KUKA KRL program: Screwing_Demo.src, Screwing_Demo.dat

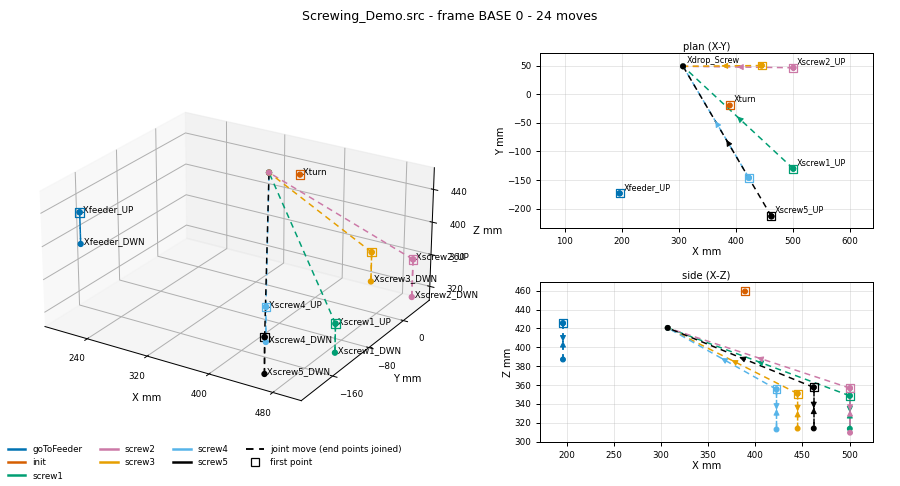
[picture p0: tool path of Screwing_Demo.src in frame BASE 0, 24 of 28 moves have a stored position in this frame; points joined in program order, loops and branches not executed]
--- Screwing_Demo.src ---
&ACCESS RVP
&REL 1
&PARAM DISKPATH = KRC:\R1\Program
DEF Screwing_Demo( )
INTERRUPT DECL 3 WHEN aiVacuumInput < 0.230 DO screwDropInterrupt()
;FOLD INI;%{PE}
  ;FOLD BASISTECH INI
    GLOBAL INTERRUPT DECL 3 WHEN $STOPMESS==TRUE DO IR_STOPM ( )
    INTERRUPT ON 3
    BAS (#INITMOV,0 )
  ;ENDFOLD (BASISTECH INI)
;FOLD SPOTTECH INI
USERSPOT(#INIT)
;ENDFOLD (SPOTTECH INI)
;FOLD GRIPPERTECH INI
USER_GRP(0,DUMMY,DUMMY,GDEFAULT)
;ENDFOLD (GRIPPERTECH INI)
  ;FOLD USER INI
    ;Make your modifications here

  ;ENDFOLD (USER INI)
;ENDFOLD (INI)
;FOLD PTP HOME  Vel= 100 % DEFAULT;%{PE}%MKUKATPBASIS,%CMOVE,%VPTP,%P 1:PTP, 2:HOME, 3:, 5:100, 7:DEFAULT
$BWDSTART = FALSE
PDAT_ACT=PDEFAULT
FDAT_ACT=FHOME
BAS (#PTP_PARAMS,100 )
$H_POS=XHOME
PTP  XHOME
;ENDFOLD
num_state_machine = 1
LOOP
 SWITCH num_state_machine
  CASE init_state
    init()
  CASE screw1_state
   resetOutputs()
   goToFeeder()
   screw1()
  CASE screw2_state
   resetOutputs()
   goToFeeder()
   screw2()
  CASE screw3_state
   resetOutputs()
   goToFeeder()
   screw3()
  CASE screw4_state
   resetOutputs()
   goToFeeder()
   screw4()
  CASE screw5_state
   resetOutputs()
   goToFeeder()
   screw5()
  CASE error_state
   EXIT
 ENDSWITCH
ENDLOOP
END
DEF screwingProcess()
 $ACC.CP = 1
 $VEL.CP = 1
 INTERRUPT ON
 LIN_REL { Z - 15}
 WAIT FOR TRUE
END
DEF goToFeeder()
;FOLD PTP feeder_UP Vel=100 % PDAT2 Tool[1] Base[0];%{PE}%R 8.3.40,%MKUKATPBASIS,%CMOVE,%VPTP,%P 1:PTP, 2:feeder_UP, 3:, 5:100, 7:PDAT2
$BWDSTART=FALSE
PDAT_ACT=PPDAT2
FDAT_ACT=Ffeeder_UP
BAS(#PTP_PARAMS,100)
PTP Xfeeder_UP
;ENDFOLD
 setVel()
;FOLD PTP feeder_DWN Vel=100 % PDAT3 Tool[1] Base[0];%{PE}%R 8.3.40,%MKUKATPBASIS,%CMOVE,%VPTP,%P 1:PTP, 2:feeder_DWN, 3:, 5:100, 7:PDAT3
$BWDSTART=FALSE
PDAT_ACT=PPDAT3
FDAT_ACT=Ffeeder_DWN
BAS(#PTP_PARAMS,100)
PTP Xfeeder_DWN
;ENDFOLD
 Vacuum_ON = TRUE
 ANIN ON vacuumValue = 1.0 * aiVacuumInput
 WAIT FOR vacuumValue >= 0.23
 ANIN OFF aiVacuumInput
;FOLD PTP feeder_UP Vel=100 % PDAT4 Tool[1] Base[0];%{PE}%R 8.3.40,%MKUKATPBASIS,%CMOVE,%VPTP,%P 1:PTP, 2:feeder_UP, 3:, 5:100, 7:PDAT4
$BWDSTART=FALSE
PDAT_ACT=PPDAT4
FDAT_ACT=Ffeeder_UP
BAS(#PTP_PARAMS,100)
PTP Xfeeder_UP
;ENDFOLD
END
DEF screwInterruptOK()
 INTERRUPT OFF
 BRAKE
 LIN $POS_INT
 RESUME
END
DEF screwInterruptNOK()
 INTERRUPT OFF
 BRAKE
 LIN $POS_INT
 RESUME
END
DEF setVel()
 $OV_PRO = 10
 $ACC.CP = 2
 $VEL.CP = 2
END
DEF setPathVel()
 $OV_PRO = 60
END
DEF init()
 setPathVel()
;FOLD PTP turn Vel=100 % PDAT1 Tool[1] Base[0];%{PE}%R 8.3.40,%MKUKATPBASIS,%CMOVE,%VPTP,%P 1:PTP, 2:turn, 3:, 5:100, 7:PDAT1
$BWDSTART=FALSE
PDAT_ACT=PPDAT1
FDAT_ACT=Fturn
BAS(#PTP_PARAMS,100)
PTP Xturn
;ENDFOLD
 num_state_machine = screw1_state
END
DEF resetOutputs()
 doResetProg = TRUE
 WAIT SEC 0.024
 doStartScrewing = FALSE
 doResetProg = FALSE
END
DEF screw1()
INTERRUPT DECL 1 WHEN diScrewOK DO screwInterruptOK()
INTERRUPT DECL 2 WHEN diScrewNOK DO screwInterruptNOK()
setPathVel()
;FOLD PTP screw1_UP Vel=100 % PDAT7 Tool[1] Base[0];%{PE}%R 8.3.40,%MKUKATPBASIS,%CMOVE,%VPTP,%P 1:PTP, 2:screw1_UP, 3:, 5:100, 7:PDAT7
$BWDSTART=FALSE
PDAT_ACT=PPDAT7
FDAT_ACT=Fscrew1_UP
BAS(#PTP_PARAMS,100)
PTP Xscrew1_UP
;ENDFOLD
setVel()
;FOLD PTP screw1_DWN Vel=100 % PDAT6 Tool[1] Base[0];%{PE}%R 8.3.40,%MKUKATPBASIS,%CMOVE,%VPTP,%P 1:PTP, 2:screw1_DWN, 3:, 5:100, 7:PDAT6
$BWDSTART=FALSE
PDAT_ACT=PPDAT6
FDAT_ACT=Fscrew1_DWN
BAS(#PTP_PARAMS,100)
PTP Xscrew1_DWN
;ENDFOLD
 doStartScrewing = TRUE
 screwingProcess()
 Vacuum_ON = FALSE
setPathVel()
;FOLD PTP screw1_UP Vel=100 % PDAT8 Tool[1] Base[0];%{PE}%R 8.3.40,%MKUKATPBASIS,%CMOVE,%VPTP,%P 1:PTP, 2:screw1_UP, 3:, 5:100, 7:PDAT8
$BWDSTART=FALSE
PDAT_ACT=PPDAT8
FDAT_ACT=Fscrew1_UP
BAS(#PTP_PARAMS,100)
PTP Xscrew1_UP
;ENDFOLD
;FOLD PTP drop_Screw Vel=100 % PDAT5 Tool[1] Base[0];%{PE}%R 8.3.40,%MKUKATPBASIS,%CMOVE,%VPTP,%P 1:PTP, 2:drop_Screw, 3:, 5:100, 7:PDAT5
$BWDSTART=FALSE
PDAT_ACT=PPDAT5
FDAT_ACT=Fdrop_Screw
BAS(#PTP_PARAMS,100)
PTP Xdrop_Screw
;ENDFOLD
 num_state_machine = screw2_state
END
DEF screw2()
setPathVel()
;FOLD PTP screw2_UP Vel=100 % PDAT10 Tool[1] Base[0];%{PE}%R 8.3.40,%MKUKATPBASIS,%CMOVE,%VPTP,%P 1:PTP, 2:screw2_UP, 3:, 5:100, 7:PDAT10
$BWDSTART=FALSE
PDAT_ACT=PPDAT10
FDAT_ACT=Fscrew2_UP
BAS(#PTP_PARAMS,100)
PTP Xscrew2_UP
;ENDFOLD
setVel()
;FOLD PTP screw2_DWN Vel=100 % PDAT9 Tool[1] Base[0];%{PE}%R 8.3.40,%MKUKATPBASIS,%CMOVE,%VPTP,%P 1:PTP, 2:screw2_DWN, 3:, 5:100, 7:PDAT9
$BWDSTART=FALSE
PDAT_ACT=PPDAT9
FDAT_ACT=Fscrew2_DWN
BAS(#PTP_PARAMS,100)
PTP Xscrew2_DWN
;ENDFOLD
 doStartScrewing = TRUE
 screwingProcess()
 Vacuum_ON = FALSE
setPathVel()
;FOLD PTP screw2_UP Vel=100 % PDAT11 Tool[1] Base[0];%{PE}%R 8.3.40,%MKUKATPBASIS,%CMOVE,%VPTP,%P 1:PTP, 2:screw2_UP, 3:, 5:100, 7:PDAT11
$BWDSTART=FALSE
PDAT_ACT=PPDAT11
FDAT_ACT=Fscrew2_UP
BAS(#PTP_PARAMS,100)
PTP Xscrew2_UP
;ENDFOLD
;FOLD PTP drop_Screw Vel=100 % PDAT12 Tool[1] Base[0];%{PE}%R 8.3.40,%MKUKATPBASIS,%CMOVE,%VPTP,%P 1:PTP, 2:drop_Screw, 3:, 5:100, 7:PDAT12
$BWDSTART=FALSE
PDAT_ACT=PPDAT12
FDAT_ACT=Fdrop_Screw
BAS(#PTP_PARAMS,100)
PTP Xdrop_Screw
;ENDFOLD
 num_state_machine = screw3_state
END
DEF screw3()
 setPathVel()
;FOLD PTP screw3_UP Vel=100 % PDAT13 Tool[1] Base[0];%{PE}%R 8.3.40,%MKUKATPBASIS,%CMOVE,%VPTP,%P 1:PTP, 2:screw3_UP, 3:, 5:100, 7:PDAT13
$BWDSTART=FALSE
PDAT_ACT=PPDAT13
FDAT_ACT=Fscrew3_UP
BAS(#PTP_PARAMS,100)
PTP Xscrew3_UP
;ENDFOLD
 setVel()
;FOLD PTP screw3_DWN Vel=100 % PDAT14 Tool[1] Base[0];%{PE}%R 8.3.40,%MKUKATPBASIS,%CMOVE,%VPTP,%P 1:PTP, 2:screw3_DWN, 3:, 5:100, 7:PDAT14
$BWDSTART=FALSE
PDAT_ACT=PPDAT14
FDAT_ACT=Fscrew3_DWN
BAS(#PTP_PARAMS,100)
PTP Xscrew3_DWN
;ENDFOLD
 doStartScrewing = TRUE
 screwingProcess()
 Vacuum_ON = FALSE
 setPathVel()
;FOLD PTP screw3_UP Vel=100 % PDAT15 Tool[1] Base[0];%{PE}%R 8.3.40,%MKUKATPBASIS,%CMOVE,%VPTP,%P 1:PTP, 2:screw3_UP, 3:, 5:100, 7:PDAT15
$BWDSTART=FALSE
PDAT_ACT=PPDAT15
FDAT_ACT=Fscrew3_UP
BAS(#PTP_PARAMS,100)
PTP Xscrew3_UP
;ENDFOLD
;FOLD PTP drop_Screw Vel=100 % PDAT16 Tool[1] Base[0];%{PE}%R 8.3.40,%MKUKATPBASIS,%CMOVE,%VPTP,%P 1:PTP, 2:drop_Screw, 3:, 5:100, 7:PDAT16
$BWDSTART=FALSE
PDAT_ACT=PPDAT16
FDAT_ACT=Fdrop_Screw
BAS(#PTP_PARAMS,100)
PTP Xdrop_Screw
;ENDFOLD
 num_state_machine = screw4_state
END
DEF screw4()
 setPathVel()
;FOLD PTP screw4_UP Vel=100 % PDAT18 Tool[1] Base[0];%{PE}%R 8.3.40,%MKUKATPBASIS,%CMOVE,%VPTP,%P 1:PTP, 2:screw4_UP, 3:, 5:100, 7:PDAT18
$BWDSTART=FALSE
PDAT_ACT=PPDAT18
FDAT_ACT=Fscrew4_UP
BAS(#PTP_PARAMS,100)
PTP Xscrew4_UP
;ENDFOLD
 setVel()
;FOLD PTP screw4_DWN Vel=100 % PDAT17 Tool[1] Base[0];%{PE}%R 8.3.40,%MKUKATPBASIS,%CMOVE,%VPTP,%P 1:PTP, 2:screw4_DWN, 3:, 5:100, 7:PDAT17
$BWDSTART=FALSE
PDAT_ACT=PPDAT17
FDAT_ACT=Fscrew4_DWN
BAS(#PTP_PARAMS,100)
PTP Xscrew4_DWN
;ENDFOLD
 doStartScrewing = TRUE
 screwingProcess()
 Vacuum_ON = FALSE
 setPathVel()
;FOLD PTP screw4_UP Vel=100 % PDAT19 Tool[1] Base[0];%{PE}%R 8.3.40,%MKUKATPBASIS,%CMOVE,%VPTP,%P 1:PTP, 2:screw4_UP, 3:, 5:100, 7:PDAT19
$BWDSTART=FALSE
PDAT_ACT=PPDAT19
FDAT_ACT=Fscrew4_UP
BAS(#PTP_PARAMS,100)
PTP Xscrew4_UP
;ENDFOLD
;FOLD PTP drop_Screw Vel=100 % PDAT20 Tool[1] Base[0];%{PE}%R 8.3.40,%MKUKATPBASIS,%CMOVE,%VPTP,%P 1:PTP, 2:drop_Screw, 3:, 5:100, 7:PDAT20
$BWDSTART=FALSE
PDAT_ACT=PPDAT20
FDAT_ACT=Fdrop_Screw
BAS(#PTP_PARAMS,100)
PTP Xdrop_Screw
;ENDFOLD
 num_state_machine = screw5_state
END
DEF screw5()
 setPathVel()
;FOLD PTP screw5_UP Vel=100 % PDAT21 Tool[1] Base[0];%{PE}%R 8.3.40,%MKUKATPBASIS,%CMOVE,%VPTP,%P 1:PTP, 2:screw5_UP, 3:, 5:100, 7:PDAT21
$BWDSTART=FALSE
PDAT_ACT=PPDAT21
FDAT_ACT=Fscrew5_UP
BAS(#PTP_PARAMS,100)
PTP Xscrew5_UP
;ENDFOLD
 setVel()
;FOLD PTP screw5_DWN Vel=100 % PDAT22 Tool[1] Base[0];%{PE}%R 8.3.40,%MKUKATPBASIS,%CMOVE,%VPTP,%P 1:PTP, 2:screw5_DWN, 3:, 5:100, 7:PDAT22
$BWDSTART=FALSE
PDAT_ACT=PPDAT22
FDAT_ACT=Fscrew5_DWN
BAS(#PTP_PARAMS,100)
PTP Xscrew5_DWN
;ENDFOLD
 doStartScrewing = TRUE
 screwingProcess()
 Vacuum_ON = FALSE
 setPathVel()
;FOLD PTP screw5_UP Vel=100 % PDAT23 Tool[1] Base[0];%{PE}%R 8.3.40,%MKUKATPBASIS,%CMOVE,%VPTP,%P 1:PTP, 2:screw5_UP, 3:, 5:100, 7:PDAT23
$BWDSTART=FALSE
PDAT_ACT=PPDAT23
FDAT_ACT=Fscrew5_UP
BAS(#PTP_PARAMS,100)
PTP Xscrew5_UP
;ENDFOLD
;FOLD PTP drop_Screw Vel=100 % PDAT24 Tool[1] Base[0];%{PE}%R 8.3.40,%MKUKATPBASIS,%CMOVE,%VPTP,%P 1:PTP, 2:drop_Screw, 3:, 5:100, 7:PDAT24
$BWDSTART=FALSE
PDAT_ACT=PPDAT24
FDAT_ACT=Fdrop_Screw
BAS(#PTP_PARAMS,100)
PTP Xdrop_Screw
;ENDFOLD
 num_state_machine = error_state
END
DEF screwDropInterrupt()


END

--- Screwing_Demo.dat ---
&ACCESS RVP
&REL 1
&PARAM DISKPATH = KRC:\R1\Program
DEFDAT  Screwing_Demo
;FOLD EXTERNAL DECLARATIONS;%{PE}%MKUKATPBASIS,%CEXT,%VCOMMON,%P
;FOLD GRIPPERTECH EXT
EXT  H50 (INT  :IN,INT  :IN,INT  :IN,GRP_TYP  :IN )
;ENDFOLD (GRIPPERTECH EXT)
;FOLD SPOTTECH EXT
EXT  USERSPOT (S_COMMAND  :IN,SPOT_TYPE  :IN )
;ENDFOLD (SPOTTECH EXT)
;FOLD BASISTECH EXT;%{PE}%MKUKATPBASIS,%CEXT,%VEXT,%P
EXT  BAS (BAS_COMMAND  :IN,REAL  :IN )
DECL INT SUCCESS
;ENDFOLD (BASISTECH EXT)
;FOLD USER EXT;%{E}%MKUKATPUSER,%CEXT,%VEXT,%P
;Make your modifications here

;ENDFOLD (USER EXT)
;ENDFOLD (EXTERNAL DECLARATIONS)
DECL BASIS_SUGG_T LAST_BASIS={POINT1[] "screw5_DWN              ",POINT2[] "screw5_DWN              ",CP_PARAMS[] "CPDAT0                  ",PTP_PARAMS[] "PDAT24                  ",CONT[] "                        ",CP_VEL[] "2.0                     ",PTP_VEL[] "100                     ",SYNC_PARAMS[] "SYNCDAT                 ",SPL_NAME[] "S0                      ",A_PARAMS[] "ADAT0                   "}
DECL E6POS XTURN={X 389.211578,Y -19.3848476,Z 459.194946,A -0.811496913,B -0.226166412,C -178.571426,S 2,T 42,E1 0.0,E2 0.0,E3 0.0,E4 0.0,E5 0.0,E6 0.0}
DECL FDAT Fturn={TOOL_NO 1,BASE_NO 0,IPO_FRAME #BASE,POINT2[] " ",TQ_STATE FALSE}
DECL PDAT PPDAT1={VEL 100.000,ACC 100.000,APO_DIST 100.000,GEAR_JERK 50.0000,EXAX_IGN 0}
DECL E6POS XFEEDER_UP={X 196.220749,Y -173.381210,Z 425.570679,A -0.807977498,B -0.211325377,C -179.106140,S 2,T 42,E1 0.0,E2 0.0,E3 0.0,E4 0.0,E5 0.0,E6 0.0}
DECL FDAT Ffeeder_UP={TOOL_NO 1,BASE_NO 0,IPO_FRAME #BASE,POINT2[] " ",TQ_STATE FALSE}
DECL PDAT PPDAT2={VEL 100.000,ACC 100.000,APO_DIST 100.000,GEAR_JERK 50.0000,EXAX_IGN 0}
DECL E6POS XFEEDER_DWN={X 196.220749,Y -173.381210,Z 387.040955,A -0.807977557,B -0.211325377,C -179.106140,S 2,T 42,E1 0.0,E2 0.0,E3 0.0,E4 0.0,E5 0.0,E6 0.0}
DECL FDAT Ffeeder_DWN={TOOL_NO 1,BASE_NO 0,IPO_FRAME #BASE,POINT2[] " ",TQ_STATE FALSE}
DECL PDAT PPDAT3={VEL 100.000,ACC 100.000,APO_DIST 100.000,GEAR_JERK 50.0000,EXAX_IGN 0}
DECL PDAT PPDAT4={VEL 100.000,ACC 100.000,APO_DIST 100.000,GEAR_JERK 50.0000,EXAX_IGN 0}
DECL E6POS XDROP_SCREW={X 307.259644,Y 49.1273842,Z 420.519073,A -0.809531212,B -0.208223656,C -179.109695,S 2,T 43,E1 0.0,E2 0.0,E3 0.0,E4 0.0,E5 0.0,E6 0.0}
DECL FDAT Fdrop_Screw={TOOL_NO 1,BASE_NO 0,IPO_FRAME #BASE,POINT2[] " ",TQ_STATE FALSE}
DECL PDAT PPDAT5={VEL 100.000,ACC 100.000,APO_DIST 100.000,GEAR_JERK 50.0000,EXAX_IGN 0}
DECL E6POS XSCREW1_DWN={X 500.255096,Y -130.118561,Z 313.684326,A -0.809358656,B -0.208476350,C -179.105576,S 2,T 42,E1 0.0,E2 0.0,E3 0.0,E4 0.0,E5 0.0,E6 0.0}
DECL FDAT Fscrew1_DWN={TOOL_NO 1,BASE_NO 0,IPO_FRAME #BASE,POINT2[] " ",TQ_STATE FALSE}
DECL PDAT PPDAT6={VEL 100.000,ACC 100.000,APO_DIST 100.000,GEAR_JERK 50.0000,EXAX_IGN 0}
DECL E6POS XSCREW1_UP={X 500.255096,Y -130.118546,Z 348.575531,A -0.809358537,B -0.208476380,C -179.105576,S 2,T 42,E1 0.0,E2 0.0,E3 0.0,E4 0.0,E5 0.0,E6 0.0}
DECL FDAT Fscrew1_UP={TOOL_NO 1,BASE_NO 0,IPO_FRAME #BASE,POINT2[] " ",TQ_STATE FALSE}
DECL PDAT PPDAT7={VEL 100.000,ACC 100.000,APO_DIST 100.000,GEAR_JERK 50.0000,EXAX_IGN 0}
DECL PDAT PPDAT8={VEL 100.000,ACC 100.000,APO_DIST 100.000,GEAR_JERK 50.0000,EXAX_IGN 0}
DECL E6POS Xscrew2_UP={X 500.485687,Y 46.6302452,Z 356.683380,A -0.811561167,B -0.204191223,C -179.109436,S 2,T 43,E1 0.0,E2 0.0,E3 0.0,E4 0.0,E5 0.0,E6 0.0}
DECL FDAT Fscrew2_UP={TOOL_NO 1,BASE_NO 0,IPO_FRAME #BASE,POINT2[] " ",TQ_STATE FALSE}
DECL E6POS XSCREW2_DWN={X 500.481,Y 46.6298,Z 309.442596,A -0.811565459,B -0.204192802,C -179.109451,S 2,T 43,E1 0.0,E2 0.0,E3 0.0,E4 0.0,E5 0.0,E6 0.0}
DECL FDAT Fscrew2_DWN={TOOL_NO 1,BASE_NO 0,IPO_FRAME #BASE,POINT2[] " ",TQ_STATE FALSE}
DECL PDAT PPDAT9={VEL 100.000,ACC 100.000,APO_DIST 100.000,GEAR_JERK 50.0000,EXAX_IGN 0}
DECL PDAT PPDAT10={VEL 100.000,ACC 100.000,APO_DIST 100.000,GEAR_JERK 50.0000,EXAX_IGN 0}
DECL PDAT PPDAT11={VEL 100.000,ACC 100.000,APO_DIST 100.000,GEAR_JERK 50.0000,EXAX_IGN 0}
DECL E6POS Xscrew3_UP={X 444.938904,Y 50.5139389,Z 350.931396,A -0.812189937,B -0.208805472,C -179.116608,S 2,T 43,E1 0.0,E2 0.0,E3 0.0,E4 0.0,E5 0.0,E6 0.0}
DECL FDAT Fscrew3_UP={TOOL_NO 1,BASE_NO 0,IPO_FRAME #BASE,POINT2[] " ",TQ_STATE FALSE}
DECL PDAT PPDAT12={VEL 100.000,ACC 100.000,APO_DIST 100.000,GEAR_JERK 50.0000,EXAX_IGN 0}
DECL PDAT PPDAT13={VEL 100.000,ACC 100.000,APO_DIST 100.000,GEAR_JERK 50.0000,EXAX_IGN 0}
DECL E6POS XSCREW3_DWN={X 444.932312,Y 50.5131683,Z 313.837921,A -0.812199831,B -0.208808899,C -179.116638,S 2,T 43,E1 0.0,E2 0.0,E3 0.0,E4 0.0,E5 0.0,E6 0.0}
DECL FDAT Fscrew3_DWN={TOOL_NO 1,BASE_NO 0,IPO_FRAME #BASE,POINT2[] " ",TQ_STATE FALSE}
DECL PDAT PPDAT14={VEL 100.000,ACC 100.000,APO_DIST 100.000,GEAR_JERK 50.0000,EXAX_IGN 0}
DECL PDAT PPDAT15={VEL 100.000,ACC 100.000,APO_DIST 100.000,GEAR_JERK 50.0000,EXAX_IGN 0}
DECL E6POS Xscrew4_UP={X 422.566467,Y -146.153397,Z 355.423981,A -0.813756645,B -0.209180310,C -179.120575,S 2,T 42,E1 0.0,E2 0.0,E3 0.0,E4 0.0,E5 0.0,E6 0.0}
DECL FDAT Fscrew4_UP={TOOL_NO 1,BASE_NO 0,IPO_FRAME #BASE,POINT2[] " ",TQ_STATE FALSE}
DECL PDAT PPDAT16={VEL 100.000,ACC 100.000,APO_DIST 100.000,GEAR_JERK 50.0000,EXAX_IGN 0}
DECL E6POS XSCREW4_DWN={X 422.564392,Y -146.152679,Z 312.870300,A -0.813760102,B -0.209177017,C -179.120575,S 2,T 42,E1 0.0,E2 0.0,E3 0.0,E4 0.0,E5 0.0,E6 0.0}
DECL FDAT Fscrew4_DWN={TOOL_NO 1,BASE_NO 0,IPO_FRAME #BASE,POINT2[] " ",TQ_STATE FALSE}
DECL PDAT PPDAT17={VEL 100.000,ACC 100.000,APO_DIST 100.000,GEAR_JERK 50.0000,EXAX_IGN 0}
DECL PDAT PPDAT18={VEL 100.000,ACC 100.000,APO_DIST 100.000,GEAR_JERK 50.0000,EXAX_IGN 0}
DECL PDAT PPDAT19={VEL 100.000,ACC 100.000,APO_DIST 100.000,GEAR_JERK 50.0000,EXAX_IGN 0}
DECL E6POS Xscrew5_UP={X 462.037201,Y -213.616409,Z 357.487885,A -0.813229620,B -0.209421441,C -179.118744,S 2,T 42,E1 0.0,E2 0.0,E3 0.0,E4 0.0,E5 0.0,E6 0.0}
DECL FDAT Fscrew5_UP={TOOL_NO 1,BASE_NO 0,IPO_FRAME #BASE,POINT2[] " ",TQ_STATE FALSE}
DECL PDAT PPDAT20={VEL 100.000,ACC 100.000,APO_DIST 100.000,GEAR_JERK 50.0000,EXAX_IGN 0}
DECL PDAT PPDAT21={VEL 100.000,ACC 100.000,APO_DIST 100.000,GEAR_JERK 50.0000,EXAX_IGN 0}
DECL E6POS XSCREW5_DWN={X 462.037201,Y -213.616409,Z 313.974304,A -0.813229322,B -0.209421501,C -179.118744,S 2,T 42,E1 0.0,E2 0.0,E3 0.0,E4 0.0,E5 0.0,E6 0.0}
DECL FDAT Fscrew5_DWN={TOOL_NO 1,BASE_NO 0,IPO_FRAME #BASE,POINT2[] " ",TQ_STATE FALSE}
DECL PDAT PPDAT22={VEL 100.000,ACC 100.000,APO_DIST 100.000,GEAR_JERK 50.0000,EXAX_IGN 0}
DECL PDAT PPDAT23={VEL 100.000,ACC 100.000,APO_DIST 100.000,GEAR_JERK 50.0000,EXAX_IGN 0}
DECL E6POS Xscrew6_UP={X 462.546967,Y -214.779938,Z 353.413391,A -0.813230276,B -0.209421292,C -179.118744,S 2,T 42,E1 0.0,E2 0.0,E3 0.0,E4 0.0,E5 0.0,E6 0.0}
DECL FDAT Fscrew6_UP={TOOL_NO 1,BASE_NO 0,IPO_FRAME #BASE,POINT2[] " ",TQ_STATE FALSE}
DECL PDAT PPDAT24={VEL 100.000,ACC 100.000,APO_DIST 100.000,GEAR_JERK 50.0000,EXAX_IGN 0}
ENDDAT
